Staubli VAL3: getErrorCode.pgx

public program getErrorCode(num x_nCamID (dimensions=1), num& x_nErrorCode[] (dimensions=1))
begin
  //-----------------------------------------------------------------------
  //Header begin
  //Description of program
  //  Get error code of last executed command.
  //
  //Input parameters
  //  num x_nCamID :
  //    role : camera's ID
  //
  //Output parameters
  //  num x_nErrorCode :
  //    role : error code of the last executed command
  //
  //Examples
  //  call getErrorCode(nCamID,l_nErrorCode)
  //
  //History
  //  Creation : 19-05-08 - f.Rob
  //  Modification 06-2012 - T.Caille - C.Rocchini
  //Header end
  //-----------------------------------------------------------------------
  if nLibErrorCode==0
    x_nErrorCode=cCamera[x_nCamID].nErrorCode
  else
    x_nErrorCode=nLibErrorCode
    nLibErrorCode=0
  endIf
  nCamID=x_nCamID
end
